PROGRAM SEQ_CR_PICK
VAR_INPUT
	CR_sequence		: UINT;
	CR_PickRack		: UINT :=1;
END_VAR

VAR
	process_T	: UINT; //CR Pick
	process_U	: UINT; //Place COSMO
	
	CR_racknum	: UINT;
	CR_PickNum	: UINT;
	OutBit1		: INT;
	OutBit2		: INT;
	InBit1		: INT;
	InBit2		: INT;
	Msg_CR		: STRING;
END_VAR

IF AUTO_MODE.COSMO_LOAD OR AUTO_MODE.JIGC_PICK OR AUTO_MODE.VB_PICK THEN
	RETURN;
END_IF
		
IF NOT AUTO_MODE.CR_UNLOADING AND NOT AUTO_MODE.COSMO_LOAD AND KR2.Idle THEN
	FOR CR_Picknum := 2 TO 21 BY 1 DO
		IF CR_Picknum = 14 THEN
			CONTINUE;
		END_IF
		IF GVL.CR_NextPickNum > 21 OR GVL.CR_NextPickNum < 2 OR CR_PickNum > 21 THEN
			GVL.CR_NextPickNum := 2; CR_PickNum := 2;
		END_IF
		IF GVL.CRTimer[CR_PickNum] < 1 THEN
			AUTO_MODE.CR_UNLOADING := TRUE;
			CR_PickRack := CR_PickNum;
			GVL.CR_NextPickNum := CR_PickNum + 1;
			RETURN;
		END_IF
	END_FOR
END_IF	

//return;
CASE CR_sequence OF
	0:
		AUTO_MODE.processnameCR := CONCAT(MSG.COMP_CR,MSG.ACTION_INIT);	
		LOGPROCESS( spLogComp	 := MSG.COMP_CR, 
		 			spLogAction	 := MSG.ACTION_INIT, 
		 			spLogStatus	 := MSG.STATUS_DONE,
	 	 		 	plogFlag	 := TRUE);
		process_T	:= 0;
		process_U	:= 0;
		CR_sequence := 1;
		
	// CR PICK --------------------------------------------------------------------------------------------------------------		
	1: 
		IF process_T = 0 THEN
			IF KR2.Idle AND GVL.COSMO_Ready AND AUTO_MODE.CR_UNLOADING and COOL_RACK.CR[CR_PickRack] THEN
				CASE CR_PickRack OF
					1:
//						OutBit1	:=	InBit1 				:= 6; 
//						OutBit2	:= 	InBit2 				:= 1;
//						KR2.bOutBit[OutBit1,OutBit2] 	:= TRUE;
						Msg_CR 							:= MSG.ACTION_CR1_PICK;
						AUTO_MODE.CR_PICK 				:= TRUE;
						process_T 						:= 1;
					2:
						OutBit1	:=	InBit1 				:= 6; 
						OutBit2	:= 	InBit2 				:= 2;
						KR2.bOutBit[OutBit1,OutBit2] 	:= TRUE;
						Msg_CR 							:= MSG.ACTION_CR2_PICK;
						AUTO_MODE.CR_PICK 				:= TRUE;
						process_T 						:= 1;
					3:
						OutBit1	:=	InBit1 				:= 6; 
						OutBit2	:= 	InBit2 				:= 3;
						KR2.bOutBit[OutBit1,OutBit2] 	:= TRUE;
						Msg_CR 							:= MSG.ACTION_CR3_PICK;
						AUTO_MODE.CR_PICK 				:= TRUE;
						process_T 						:= 1;
					4:
						OutBit1	:=	InBit1 				:= 6; 
						OutBit2	:= 	InBit2 				:= 4;
						KR2.bOutBit[OutBit1,OutBit2] 	:= TRUE;
						Msg_CR 							:= MSG.ACTION_CR4_PICK;
						AUTO_MODE.CR_PICK 				:= TRUE;
						process_T 						:= 1;
					5:
						OutBit1	:=	InBit1 				:= 6; 
						OutBit2	:= 	InBit2 				:= 5;
						KR2.bOutBit[OutBit1,OutBit2] 	:= TRUE;
						Msg_CR 							:= MSG.ACTION_CR5_PICK;
						AUTO_MODE.CR_PICK 				:= TRUE;
						process_T 						:= 1;
					6:
						OutBit1	:=	InBit1 				:= 6; 
						OutBit2	:= 	InBit2 				:= 6;
						KR2.bOutBit[OutBit1,OutBit2] 	:= TRUE;
						Msg_CR 							:= MSG.ACTION_CR6_PICK;
						AUTO_MODE.CR_PICK 				:= TRUE;
						process_T 						:= 1;
					7:
						OutBit1	:=	InBit1 				:= 6; 
						OutBit2	:= 	InBit2 				:= 7;
						KR2.bOutBit[OutBit1,OutBit2] 	:= TRUE;
						Msg_CR 							:= MSG.ACTION_CR7_PICK;
						AUTO_MODE.CR_PICK 				:= TRUE;
						process_T 						:= 1;
					8:
//						OutBit1	:=	InBit1 				:= 7; 
//						OutBit2	:= 	InBit2 				:= 0;
//						KR2.bOutBit[OutBit1,OutBit2] 	:= TRUE;
						Msg_CR 							:= MSG.ACTION_CR8_PICK;
						AUTO_MODE.CR_PICK 				:= TRUE;
						process_T 						:= 1;
					9:
						OutBit1	:=	InBit1 				:= 7; 
						OutBit2	:= 	InBit2 				:= 1;
						KR2.bOutBit[OutBit1,OutBit2] 	:= TRUE;
						Msg_CR 							:= MSG.ACTION_CR9_PICK;
						AUTO_MODE.CR_PICK 				:= TRUE;
						process_T 						:= 1;
					10:
						OutBit1	:=	InBit1 				:= 7; 
						OutBit2	:= 	InBit2 				:= 2;
						KR2.bOutBit[OutBit1,OutBit2] 	:= TRUE;
						Msg_CR 							:= MSG.ACTION_CR10_PICK;
						AUTO_MODE.CR_PICK 				:= TRUE;
						process_T 						:= 1;
					11:
						OutBit1	:=	InBit1 				:= 7; 
						OutBit2	:= 	InBit2 				:= 3;
						KR2.bOutBit[OutBit1,OutBit2] 	:= TRUE;
						Msg_CR 							:= MSG.ACTION_CR11_PICK;
						AUTO_MODE.CR_PICK 				:= TRUE;
						process_T 						:= 1;
					12:
						OutBit1	:=	InBit1 				:= 7; 
						OutBit2	:= 	InBit2 				:= 4;
						KR2.bOutBit[OutBit1,OutBit2] 	:= TRUE;
						Msg_CR 							:= MSG.ACTION_CR12_PICK;
						AUTO_MODE.CR_PICK 				:= TRUE;
						process_T 						:= 1;
					13:
						OutBit1	:=	InBit1 				:= 7; 
						OutBit2	:= 	InBit2 				:= 5;
						KR2.bOutBit[OutBit1,OutBit2] 	:= TRUE;
						Msg_CR 							:= MSG.ACTION_CR13_PICK;
						AUTO_MODE.CR_PICK 				:= TRUE;
						process_T 						:= 1;
					15:
//						OutBit1	:=	InBit1 				:= 7; 
//						OutBit2	:= 	InBit2 				:= 6;
//						KR2.bOutBit[OutBit1,OutBit2] 	:= TRUE;
						Msg_CR 							:= MSG.ACTION_CR15_PICK;
						AUTO_MODE.CR_PICK 				:= TRUE;
						process_T 						:= 1;
					16:
						OutBit1	:=	InBit1 				:= 7; 
						OutBit2	:= 	InBit2 				:= 7;
						KR2.bOutBit[OutBit1,OutBit2] 	:= TRUE;
						Msg_CR 							:= MSG.ACTION_CR16_PICK;
						AUTO_MODE.CR_PICK 				:= TRUE;
						process_T 						:= 1;
					17:
						OutBit1	:=	InBit1 				:= 8; 
						OutBit2	:= 	InBit2 				:= 0;
						KR2.bOutBit[OutBit1,OutBit2] 	:= TRUE;
						Msg_CR 							:= MSG.ACTION_CR17_PICK;
						AUTO_MODE.CR_PICK 				:= TRUE;
						process_T 						:= 1;
					18:
						OutBit1	:=	InBit1 				:= 8; 
						OutBit2	:= 	InBit2 				:= 1;
						KR2.bOutBit[OutBit1,OutBit2] 	:= TRUE;
						Msg_CR 							:= MSG.ACTION_CR18_PICK;
						AUTO_MODE.CR_PICK 				:= TRUE;
						process_T 						:= 1;
					19:
						OutBit1	:=	InBit1 				:= 8; 
						OutBit2	:= 	InBit2 				:= 2;
						KR2.bOutBit[OutBit1,OutBit2] 	:= TRUE;
						Msg_CR 							:= MSG.ACTION_CR19_PICK;
						AUTO_MODE.CR_PICK 				:= TRUE;
						process_T 						:= 1;
					20:
						OutBit1	:=	InBit1 				:= 8; 
						OutBit2	:= 	InBit2 				:= 3;
						KR2.bOutBit[OutBit1,OutBit2] 	:= TRUE;
						Msg_CR 							:= MSG.ACTION_CR20_PICK;
						AUTO_MODE.CR_PICK 				:= TRUE;
						process_T 						:= 1;
					21:
						OutBit1	:=	InBit1 				:= 8; 
						OutBit2	:= 	InBit2 				:= 4;
						KR2.bOutBit[OutBit1,OutBit2] 	:= TRUE;
						Msg_CR 							:= MSG.ACTION_CR21_PICK;
						AUTO_MODE.CR_PICK 				:= TRUE;
						process_T 						:= 1;
				END_CASE
				
				AUTO_MODE.processnameCR := CONCAT(MSG.COMP_CR,Msg_CR);
				AUTO_MODE.processnameCR := CONCAT(AUTO_MODE.processnameCR,MSG.STATUS_RUN);
				LOGPROCESS( spLogComp	 := MSG.COMP_CR, 
							spLogAction	 := Msg_CR, 
							spLogStatus	 := MSG.STATUS_RUN,
							plogFlag	 := TRUE);
			END_IF
		ELSIF process_T = 1 THEN
			KR2.bOutBit[OutBit1,OutBit2] := TRUE;
			IF KR2.bInBit[InBit1,InBit2] THEN
				KR2.bOutBit[OutBit1,OutBit2] := FALSE;	
				AUTO_MODE.processnameCR := CONCAT(MSG.COMP_CR,MSG.ACTION_CR_PICK);
				AUTO_MODE.processnameCR := CONCAT(AUTO_MODE.processnameCR,MSG.STATUS_ACK);
				LOGPROCESS( spLogComp	 := MSG.COMP_CR, 
							spLogAction	 := MSG.ACTION_CR_PICK, 
							spLogStatus	 := MSG.STATUS_ACK,
							plogFlag	 := TRUE);
				process_T := 2;
				RETURN;
			END_IF	
		ELSIF process_T = 2 THEN
			KR2.bOutBit[OutBit1,OutBit2] := FALSE;
			IF NOT KR2.bInBit[InBit1,InBit2] THEN
				AUTO_MODE.processnameCR := CONCAT(MSG.COMP_CR,MSG.ACTION_CR_PICK);
				AUTO_MODE.processnameCR := CONCAT(AUTO_MODE.processnameCR,MSG.STATUS_DONE);
				LOGPROCESS( spLogComp	 := MSG.COMP_CR, 
							spLogAction	 := MSG.ACTION_CR_PICK, 
							spLogStatus	 := MSG.STATUS_DONE,
							plogFlag	 := TRUE);
				process_T:= 3;
				RETURN;
			END_IF	
		ELSIF process_T = 3 THEN
			IF KR2.Idle AND GVL.COSMO_Ready THEN
				AUTO_MODE.processnameCR := CONCAT(MSG.COMP_CR,MSG.ACTION_CR_PICK);
				AUTO_MODE.processnameCR := CONCAT(AUTO_MODE.processnameCR,MSG.STATUS_COMP);
				LOGPROCESS( spLogComp	 := MSG.COMP_CR, 
							spLogAction	 := MSG.ACTION_CR_PICK, 
							spLogStatus	 := MSG.STATUS_COMP,
							plogFlag	 := TRUE);
				process_T := 4;
				CR_sequence := 2;
				AUTO_MODE.next_step := FALSE;
				GVL.CRTimer[CR_PickNum] := GVL.iCooling_Time;
			END_IF
		END_IF
	
	// PLACE COSMO --------------------------------------------------------------------------------------------------------------		
	2: 
		IF process_U = 0 THEN
			IF KR2.Idle AND GVL.COSMO_Ready THEN
//				KR2.PLC_O_D3.3 := TRUE; //203
				KR2.bOutBit[3,3] := TRUE;
				AUTO_MODE.processnameCR := CONCAT(MSG.COMP_CR,MSG.ACTION_COSMO_PLACE);
				AUTO_MODE.processnameCR := CONCAT(AUTO_MODE.processnameCR,MSG.STATUS_RUN);
				LOGPROCESS( spLogComp	 := MSG.COMP_CR, 
							spLogAction	 := MSG.ACTION_COSMO_PLACE, 
							spLogStatus	 := MSG.STATUS_RUN,
							plogFlag	 := TRUE);
				process_U := 1;
				RETURN;
			END_IF
		ELSIF process_U = 1 THEN
//			KR2.PLC_O_D3.3 := TRUE; //203
			KR2.bOutBit[3,3] := TRUE;
			IF KR2.bInBit[3,3] THEN
//				KR2.PLC_O_D3.3 := FALSE; //203
				KR2.bOutBit[3,3] := FALSE;
				AUTO_MODE.processnameCR := CONCAT(MSG.COMP_CR,MSG.ACTION_COSMO_PLACE);
				AUTO_MODE.processnameCR := CONCAT(AUTO_MODE.processnameCR,MSG.STATUS_ACK);
				LOGPROCESS( spLogComp	 := MSG.COMP_CR, 
							spLogAction	 := MSG.ACTION_COSMO_PLACE, 
							spLogStatus	 := MSG.STATUS_ACK,
							plogFlag	 := TRUE);
				process_U := 2;
				RETURN;
			END_IF
		ELSIF process_U = 2 THEN
//			KR2.PLC_O_D3.3 := FALSE; //203
			KR2.bOutBit[3,3] := FALSE;
			IF NOT KR2.bInBit[3,3] THEN
				AUTO_MODE.processnameCR := CONCAT(MSG.COMP_CR,MSG.ACTION_COSMO_PLACE);
				AUTO_MODE.processnameCR := CONCAT(AUTO_MODE.processnameCR,MSG.STATUS_DONE);
				LOGPROCESS( spLogComp	 := MSG.COMP_CR, 
							spLogAction	 := MSG.ACTION_COSMO_PLACE, 
							spLogStatus	 := MSG.STATUS_DONE,
							plogFlag	 := TRUE);
				IF NOT GVL.COSMO_Ready THEN
					GVL.COSMO_Run := TRUE;
					AUTO_MODE.processnameCR := 'COSMO - (RUN)';
				END_IF
				process_U := 3;
				RETURN;
			END_IF
		ELSIF process_U = 3 THEN
			IF KR2.Idle THEN
				AUTO_MODE.processnameCR := CONCAT(MSG.COMP_CR,MSG.ACTION_COSMO_PLACE);
				AUTO_MODE.processnameCR := CONCAT(AUTO_MODE.processnameCR,MSG.STATUS_COMP);
				LOGPROCESS( spLogComp	 := MSG.COMP_CR, 
							spLogAction	 := MSG.ACTION_COSMO_PLACE, 
							spLogStatus	 := MSG.STATUS_COMP,
							plogFlag	 := TRUE);
				process_U := 4;
				CR_sequence := 3;
				AUTO_MODE.COSMO_LOAD	:= TRUE;
				AUTO_MODE.COSMO_RUN 	:= TRUE;
				AUTO_MODE.CR_PICK 		:= FALSE;
				AUTO_MODE.next_step 	:= FALSE;
				AUTO_MODE.processnameCR := CONCAT(MSG.COMP_CR,MAIN.fb_TimeStamp.SystemTime);
				AUTO_MODE.processnameCR := CONCAT(AUTO_MODE.processnameCR,MSG.STATUS_END);
				LOGPROCESS( spLogComp	 := MSG.COMP_CR, 
							spLogAction	 := MSG.ACTION_CR_TO_COSMO, 
							spLogStatus	 := MSG.STATUS_END,
							plogFlag	 := TRUE);
			END_IF
		END_IF
		
	// END -------------------------------------------------------------------------------------------------------------	
	3:
		CR_sequence := 0;
		AUTO_MODE.next_step := FALSE;
END_CASE

END_PROGRAM

(* stored: Version 1.1.0.1, ProductVersion 3.1.4024.12
   POU SEQ_CR_PICK: Id {96825f8c-74be-47cc-a7f8-f20f13d897f8}, SpecialFunc None *)
